FUNCTION_BLOCK CylControlILAdpOL (* Composite Function Block Type *)
  (* Standard: 61499-2 *)
  (* Version 0.0, 7/14/2023, valeriy, nxtControl GmBH, template *)
  PACKAGE Main;
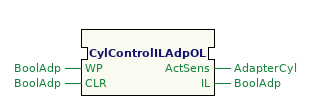
  SOCKETS
    WP : BoolAdp;
    CLR : BoolAdp;
  END_SOCKETS
  PLUGS
    ActSens : AdapterCyl;
    IL : BoolAdp;
  END_PLUGS
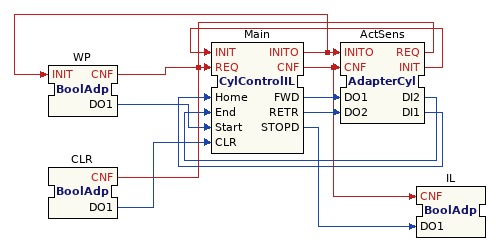
  FBS
    Main : CylControlIL;
  END_FBS
  EVENT_CONNECTIONS
    WP.CNF TO Main.REQ;
    Main.INITO TO ActSens.INITO;
    Main.CNF TO ActSens.CNF;
    Main.INITO TO WP.INIT;
    ActSens.REQ TO Main.REQ;
    ActSens.INIT TO Main.INIT;
    CLR.CNF TO Main.REQ;
    Main.CNF TO IL.CNF;
  END_CONNECTIONS
  DATA_CONNECTIONS
    WP.DO1 TO Main.Start;
    Main.FWD TO ActSens.DO1;
    Main.RETR TO ActSens.DO2;
    ActSens.DI2 TO Main.End;
    ActSens.DI1 TO Main.Home;
    CLR.DO1 TO Main.CLR;
    Main.STOPD TO IL.DO1;
  END_CONNECTIONS
END_FUNCTION_BLOCK
